TYPE
    ST_Indicator_Status : STRUCT
        On       : BOOL;
        Off      : BOOL;
        Flashing : BOOL;
    END_STRUCT
END_TYPE

(* stored: Version 1.1.0.1
   DUT ST_Indicator_Status: Id {7f662d87-a5e6-4516-86b9-34bc91b40cf7} *)
